# EPICS autosave request: iocBoot/iocDxpLinux/auto_settings.req
file "mca_settings.req",                P=dxpLinux:, M=dxp_adc1
file "dxp_settings.req",                P=dxpLinux:, R=dxp1
